# EPICS autosave request: support/ebrick/2-2-3/iocBoot/iocebrick/autosave/ccdParam_settings.req
$(P)$(E)$(T):name
